{attribute addProperty BoxType "EK1100-0000-0018"}
{attribute addProperty Id "Beckhoff_EJ6xxxEK1122Beckhoff_EJ6xxxEK1122_30779985162A_0001_EJ6002_0000_0016EJ6002_880A624E850106.25A_0002_EJ6224_0000_0016EJ6224_3990B4B417822.25A_0003_EJ6224_0090_0016EJ6224_3990B4B417822.25"}
{attribute addProperty CRC "2699412160"}
{attribute addProperty SizeInBites "1222"}
{attribute addProperty SizeInBytes "152.75"}
TYPE Beckhoff_EJ6xxx_A0E5C2C0 EXTENDS EK1100_179A0949 :
STRUCT
	{attribute addProperty Name "Beckhoff_EJ6xxxEK1122"}
	Beckhoff_EJ6xxxEK1122 : Beckhoff_EJ6xxxEK1122_30779985;
	{attribute addProperty Name "A_0001_EJ6002_0000_0016"}
	A_0001_EJ6002_0000_0016 : EJ6002_880A624E;
	{attribute addProperty Name "A_0002_EJ6224_0000_0016"}
	A_0002_EJ6224_0000_0016 : EJ6224_3990B4B4;
	{attribute addProperty Name "A_0003_EJ6224_0090_0016"}
	A_0003_EJ6224_0090_0016 : EJ6224_3990B4B4;
END_STRUCT
END_TYPE

(* stored: Version 1.2.0.0, ProductVersion 3.1.4024.9
   DUT Beckhoff_EJ6xxx_A0E5C2C0: Id {2de2a805-613d-457d-adaf-b9963cce65b7} *)
